{attribute 'linkalways'} 
{attribute 'no_explicit_call' := 'This FB is a CLASS and must be accessed using methods or properties'}
{attribute 'enable_dynamic_creation'}
FUNCTION_BLOCK _REAL EXTENDS NumericDatatypeBase
VAR
	localData : REAL;
	activeData : REFERENCE TO REAL REF= localData;
END_VAR

PROPERTY PUBLIC Address : PVOID
GET
Address := ADR(activeData);
END_GET
END_PROPERTY

METHOD PUBLIC ClearReference
VAR_INPUT
END_VAR
activeData REF= localData;
END_METHOD

METHOD PUBLIC Clone : I_Datatype
VAR
    pClone : POINTER TO _REAL;
END_VAR
pClone := __NEW(_REAL(InitialValue := Value));
Clone := pClone^;
END_METHOD

METHOD FB_init : BOOL
VAR_INPUT
	bInitRetains : BOOL; // if TRUE, the retain variables are initialized (warm start / cold start)
	bInCopyCode : BOOL;  // if TRUE, the instance afterwards gets moved into the copy code (online change)
	InitialValue : REAL;
END_VAR
localData := InitialValue;
END_METHOD

PROPERTY PUBLIC IsEven : BOOL
GET
IsEven := FALSE;
END_GET
END_PROPERTY

PROPERTY PUBLIC IsFloat : BOOL
GET
IsFloat := TRUE;
END_GET
END_PROPERTY

PROPERTY PUBLIC IsOdd : BOOL
GET
IsOdd := FALSE;
END_GET
END_PROPERTY

PROPERTY PUBLIC IsSigned : BOOL
GET
IsSigned := TRUE;
END_GET
END_PROPERTY

METHOD PUBLIC MakeReferenceTo
VAR_INPUT
	ReferenceTarget : REFERENCE TO REAL;
END_VAR
activeData REF= ReferenceTarget;
END_METHOD

PROPERTY PUBLIC MaxValue : REAL
GET
MaxValue :=  DatatypeLimits.REAL_MAX_VALUE;
END_GET
END_PROPERTY

PROPERTY PUBLIC MinValue : REAL
GET
MinValue := DatatypeLimits.REAL_MIN_VALUE;
END_GET
END_PROPERTY

METHOD PROTECTED SerializeMaxValue
VAR_INPUT
	Serializer : I_Serializer;
END_VAR
Serializer.AddReal(MaxValue);
END_METHOD

METHOD PROTECTED SerializeMinValue
VAR_INPUT
	Serializer : I_Serializer;
END_VAR
Serializer.AddReal(MinValue);
END_METHOD

METHOD PUBLIC SerializeWith
VAR_INPUT
	Serializer : I_Serializer;
END_VAR
Serializer.AddReal(activeData);
END_METHOD

PROPERTY PUBLIC Size : UDINT
GET
Size := SIZEOF(activeData);
END_GET
END_PROPERTY

METHOD TryDeserializeFrom : BOOL
VAR_INPUT
	Deserializer : I_Deserializer;
	Feedback : I_DeserializerFeedback;
END_VAR
TryDeserializeFrom := Deserializer.TryGetReal(activeData, Feedback);
END_METHOD

METHOD TryMakeReferenceTo : BOOL
VAR_INPUT
	Target : I_Datatype;
END_VAR
VAR
	pTargetData : POINTER TO REAL;
END_VAR
IF NOT IsEquivalentTo(Target) THEN
	RETURN;
END_IF

pTargetData := Target.Address;
activeData REF= pTargetData^;
TryMakeReferenceTo := TRUE;
END_METHOD

PROPERTY PUBLIC TypeName : T_MAXSTRING
GET
TypeName := 'REAL';
END_GET
END_PROPERTY

PROPERTY PUBLIC Value : REFERENCE TO REAL
GET
Value REF= activeData;
END_GET
END_PROPERTY

END_FUNCTION_BLOCK

(* stored: Version 1.1.0.1, ProductVersion 3.1.4024.13
   POU _REAL: Id {af81a63e-8d6e-4e13-82c4-cea7a6a90fcc}, SpecialFunc None
   Folder Constructor: Id {772be0a8-5b8f-4e97-9a1e-ddfc70bfd684}
   Folder Protected: Id {73a7d6bc-5823-0be5-370f-c68c882f46ad}
   Property Address: Id {96c3b1ca-d315-4278-96e9-0a429a295678}
   Get Get: Id {754c870a-6bb6-4697-8ddd-bd5b96430ae2}
   Method ClearReference: Id {5a53fbcc-fd2b-4e2e-9caa-3190887e7155}
   Method Clone: Id {90aecf76-4048-4bc3-9eb5-50d3436ab256}
   Method FB_init: Id {10e670a3-d031-4cd0-9a95-29ca188d2cf3}
   Property IsEven: Id {f3c95207-e52d-0b33-2b8c-6a386092c932}
   Get Get: Id {bc8920a8-316b-05aa-2f51-9b7748d798e8}
   Property IsFloat: Id {998b1d60-f10c-42fb-b209-cf23d7265113}
   Get Get: Id {be19ae7d-1782-4f2a-8715-2bfe73b1c92e}
   Property IsOdd: Id {5637e9ea-f0b6-0afe-0d94-d5b5f8d6839c}
   Get Get: Id {2ea49729-5bdd-0763-18c2-5ef05ee16ce7}
   Property IsSigned: Id {3be66bb9-ae86-4afe-89e5-9b879754e616}
   Get Get: Id {974598cf-ac7c-4920-951c-6aab2b8875e7}
   Method MakeReferenceTo: Id {24ff8ff5-2ca9-4a92-be6b-dba730fe012e}
   Property MaxValue: Id {37b42ba5-de75-0c5b-301a-c6dcda945a06}
   Get Get: Id {0ba03488-d39d-0fcb-1485-9d16a1dd9e0f}
   Property MinValue: Id {3d065e58-c9c9-052f-2687-8c02cefcfcf4}
   Get Get: Id {a8c895a5-b810-0e46-2a19-cf6a2b0be73a}
   Method SerializeMaxValue: Id {612031c8-75fc-0207-032a-25dbfc4525c9}
   Method SerializeMinValue: Id {c5a80002-149b-06d0-3f45-557071d1aa7e}
   Method SerializeWith: Id {1894129e-9827-4721-ba0a-a8a7495b00b5}
   Property Size: Id {6515cbf3-317a-49f2-afb7-948583d2c3fa}
   Get Get: Id {8e118d51-4419-409f-a83e-df5dec2294d1}
   Method TryDeserializeFrom: Id {2b43cc21-9fd4-4991-8fdb-ed0d1540ae9e}
   Method TryMakeReferenceTo: Id {7513fc71-35eb-48a6-9cd9-0ee2267f620b}
   Property TypeName: Id {832138f0-f7e2-4757-9f72-fdd15365cab9}
   Get Get: Id {578ddc39-2b25-42e4-b54e-2ce92fa34cc8}
   Property Value: Id {a2c4e0f7-3179-43fc-a7d9-c01814357c52}
   Get Get: Id {da357be8-167a-4463-be1f-4d66de9ca0f7} *)
